TYPE ST_TxHmiQualisys :
STRUCT
	status : DINT;
	feedback : ST_FeedbackQualisys;
	markers : ARRAY [0..9] OF ST_3DMarkerPositionNoLabel;
END_STRUCT
END_TYPE

(* stored: Version 1.1.0.1, ProductVersion 3.1.4022.7
   DUT ST_TxHmiQualisys: Id {86f8af60-9890-43c0-a3a2-fa2652052b0e} *)
